{attribute 'linkalways'} 
{attribute 'no_explicit_call' := 'This FB is a CLASS and must be accessed using methods or properties'}
{attribute 'enable_dynamic_creation'}
FUNCTION_BLOCK Node_F_VN_MedianFilter EXTENDS VisionNode
VAR
    ipSrcImage : _ITcVnImage;
    ipDestImage : _ITcVnImage;
    nFilterSize : _UDINT(3);
    hrPrev : _HRESULT(S_OK);
	hresult : _HRESULT(S_OK);
END_VAR

METHOD PUBLIC  Clone : I_Node
VAR
	pNode : POINTER TO Node_F_VN_MedianFilter;
END_VAR
pNode := __NEW(Node_F_VN_MedianFilter);
Clone := pNode^;
END_METHOD

METHOD FB_init : BOOL
VAR_INPUT
	bInitRetains : BOOL; // if TRUE, the retain variables are initialized (warm start / cold start)
	bInCopyCode : BOOL;  // if TRUE, the instance afterwards gets moved into the copy code (online change)
END_VAR
AddInput('ipSrcImage', ipSrcImage);
AddParameter('nFilterSize', nFilterSize);
AddInput('hrPrev', hrPrev);
AddOutput('ipDestImage', ipDestImage);
AddOutput('hresult',hresult);
END_METHOD

METHOD PROTECTED OnExecute
hresult.Value := F_VN_MedianFilter(
    ipSrcImage := ipSrcImage.Value,
	ipDestImage := ipDestImage.Value,
    nFilterSize := nFilterSize.Value,
	hrPrev:= hrPrev.Value);
END_METHOD

METHOD PUBLIC PreExecutionCheck
VAR_INPUT
	Check : I_PreExecutionChecks;
END_VAR
Check.IsTrue(ipSrcImage.IsValid, 'ipSrcImage must contain an image');
Check.IsTrue(nFilterSize.isOdd, 'nFilterSize must be an odd number');
Check.IsTrue(nFilterSize.Value >= 3, 'nFilterSize must be greater than or equal to 3');

IF (nFilterSize.Value = 3) OR (nFilterSize.Value = 5) THEN
    Check.IsTrue((ipSrcImage.IsPixelDepth(8) OR
                  ipSrcImage.IsPixelDepth(16) OR
                  ipSrcImage.IsPixelDepth(32)), 'ipSrcImage must have 8, 16, or 32 bit pixel depth');
ELSE
    Check.IsTrue(ipSrcImage.IsPixelDepth(8), 'ipSrcImage must have 8 bit pixel depth');
END_IF
END_METHOD

END_FUNCTION_BLOCK

(* stored: Version 1.1.0.1, ProductVersion 3.1.4024.13
   POU Node_F_VN_MedianFilter: Id {9025872c-f06e-0aab-037a-200e6759f166}, SpecialFunc None
   Folder Constructor: Id {8ad032be-5afe-0769-263d-9cfdfdcc56cf}
   Method Clone: Id {1018fe2d-63f2-0dbc-0fa0-2c7e6fc712e1}
   Method FB_init: Id {bb2dd64d-43c2-0be6-2f89-10b36d04901d}
   Method OnExecute: Id {68ece6b6-f004-0fcf-3b18-2ff5dad40517}
   Method PreExecutionCheck: Id {45d55321-d675-0c04-1632-4ac470077b1a} *)
